{attribute 'OPC.UA.DA.StructuredType' := '1'}
TYPE ST_PumpGrundfosMagna3SetParameters :
STRUCT
	nControlModeAlgorithm : E_GrundfosMagna3ControlMode; //select controlmode: constantSpeed, constantFrequency, constantHead, constantPressure, constantDifferentialPressure, proportionalPressure, constantFlow, constantTemperature, constantLevel, autoAdapt, flowAdapt, closedLoopSensor
	nControlModeManual : E_GrundfosMagna3ControlMode;
END_STRUCT
END_TYPE

(* stored: Version 1.1.0.1, ProductVersion 3.1.4024.9
   DUT ST_PumpGrundfosMagna3SetParameters: Id {431a032e-b8d7-4d7a-861f-0bdddf47f9e7} *)
